FUNCTION_BLOCK QW_Emulated (* Composite FB wrapping other FBs *)
  (* Standard: 61499-2 *)
  (* Version 1.0, 2021-08-05, dorofeev *)
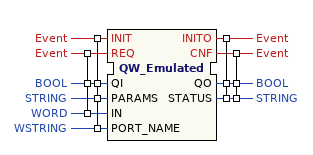
  EVENT_INPUT
    INIT WITH PARAMS, QI, PORT_NAME; (* Initialization Request *)
    REQ WITH QI, IN; (* Normal Execution Request *)
  END_EVENT
  EVENT_OUTPUT
    INITO WITH QO, STATUS; (* Initialization Confirm *)
    CNF WITH QO, STATUS; (* Execution Confirmation *)
  END_EVENT
  VAR_INPUT
    QI : BOOL; (* Input event qualifier *)
    PARAMS : STRING;
    IN : WORD;
    PORT_NAME : WSTRING;
  END_VAR
  VAR_OUTPUT
    QO : BOOL; (* Output event qualifier *)
    STATUS : STRING;
  END_VAR
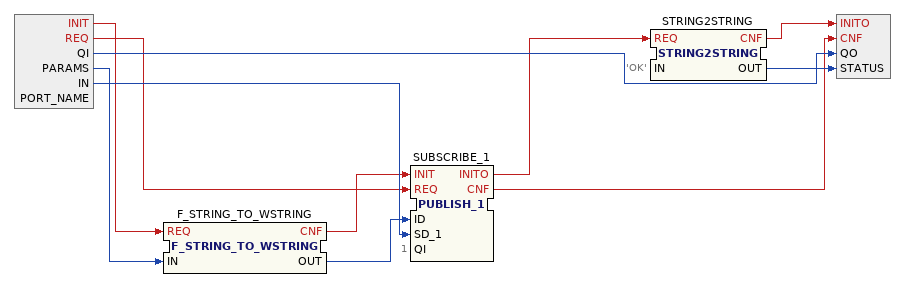
  FBS
    STRING2STRING : STRING2STRING(IN := 'OK');
    F_STRING_TO_WSTRING : F_STRING_TO_WSTRING;
    SUBSCRIBE_1 : PUBLISH_1(QI := 1);
  END_FBS
  EVENT_CONNECTIONS
    STRING2STRING.CNF TO INITO;
    INIT TO F_STRING_TO_WSTRING.REQ;
    F_STRING_TO_WSTRING.CNF TO SUBSCRIBE_1.INIT;
    SUBSCRIBE_1.INITO TO STRING2STRING.REQ;
    SUBSCRIBE_1.CNF TO CNF;
    REQ TO SUBSCRIBE_1.REQ;
  END_CONNECTIONS
  DATA_CONNECTIONS
    STRING2STRING.OUT TO STATUS;
    QI TO QO;
    PARAMS TO F_STRING_TO_WSTRING.IN;
    F_STRING_TO_WSTRING.OUT TO SUBSCRIBE_1.ID;
    IN TO SUBSCRIBE_1.SD_1;
  END_CONNECTIONS
END_FUNCTION_BLOCK
